{attribute 'pack_mode' := '2'}
TYPE ST_XPU_INFO :
STRUCT
  AllPositionsValid   : BIT;
  IdDetectionError    : BIT;
  IdDetectionValid    : BIT;
  IdDetectionActive   : BIT;

  OperationMode       : UINT;

  IdDetectionMode           : UINT;
  MoverPositionAssignement  : UINT;

  nDetectedAxisCount  : UINT;
  nExpectedAxisCount  : UINT;

  nParameterSetCount  : UINT;
  nModuleCount        : UINT;
  rRailLength         : LREAL;  
END_STRUCT
END_TYPE

(* stored: Version 1.1.0.1
   DUT ST_XPU_INFO: Id {8d4aa9a9-96cf-41e6-9d00-d152b2e6f164} *)
